{attribute addProperty BoxType "EJ2521-0224-0016"}
{attribute addProperty Id "Enable_PLSBIT10.1251OutputBIT10.1254"}
{attribute addProperty CRC "90070654"}
{attribute addProperty SizeInBites "16"}
{attribute addProperty SizeInBytes "2"}
TYPE Control_055E5E7E :
STRUCT
	{attribute addProperty Name "Enable_PLS"}
	Enable_PLS : BIT;
	{attribute 'hide'}
	reserve_1_BIT_0 : BIT;
	{attribute 'hide'}
	reserve_1_BIT_1 : BIT;
	{attribute addProperty Name "Output"}
	Output : BIT;
	{attribute 'hide'}
	reserve_2_BIT_0 : BIT;
	{attribute 'hide'}
	reserve_2_BIT_1 : BIT;
	{attribute 'hide'}
	reserve_2_BIT_2 : BIT;
	{attribute 'hide'}
	reserve_2_BIT_3 : BIT;
	{attribute 'hide'}
	reserve_3 : BYTE;
END_STRUCT
END_TYPE

(* stored: Version 1.2.0.0, ProductVersion 3.1.4024.9
   DUT Control_055E5E7E: Id {6acaf456-9d32-4077-9e9e-b01f830b0597} *)
